FUNCTION_BLOCK FB_CamAxis
VAR
  _eCheck                       : E_CHECK_STATE;
  _nErrorId                     : UDINT; // datafield for Camming error

  _AxisSlave                    : REFERENCE TO AXIS_REF;
  _AxisMaster                   : REFERENCE TO AXIS_REF;

  _fbCamInV2                    : Tc2_MC2_Camming.MC_CamIn_V2;
  _fbScalingV2                  : Tc2_MC2_Camming.MC_CamScaling_V2;
  _fbCamInfoV2                  : Tc2_MC2_Camming.MC_CamInfo_V2;

  _fbReadMotionFunction         : Tc2_MC2_Camming.MC_ReadMotionFunction;
  _fbReadMotionFunctionPoint    : Tc2_MC2_Camming.MC_ReadMotionFunctionPoint;
  _fbReadMotionFunctionValues   : Tc2_MC2_Camming.MC_ReadMotionFunctionValues;

  _fbWriteMotionFunction        : Tc2_MC2_Camming.MC_WriteMotionFunction;
  _fbWriteMotionFunctionPoint   : Tc2_MC2_Camming.MC_WriteMotionFunctionPoint;


  _stCamInfoData                : Tc2_MC2_Camming.MC_CamInfoData;

END_VAR

METHOD CamInfo : E_PROGRESS
VAR_INPUT
  Execute           : BOOL;
  CamTableID        : Tc2_MC2_Camming.MC_CAM_ID;
  AtMasterPosition  : BOOL;
  MasterPosition    : LREAL;
END_VAR
VAR_INST
  _eState           : E_PROGRESS;
  _rValue           : LREAL;
  _udiErr           : UDINT;
  _stMsg            : ST_Message;
END_VAR
IF NOT Execute THEN _eState := E_PROGRESS.INIT; END_IF

CASE _eState
OF
  E_PROGRESS.INIT:
    IF Execute 
    THEN
      memset(ADR(_stMsg),0,SIZEOF(_stMsg));
      _udiErr                       := 0;
      _rValue                       := 0;
      _eState                       := E_PROGRESS.BUSY;

      _fbCamInfoV2(
              Slave                 := _AxisSlave, 
              Execute               := FALSE, 
              CamTableID            := CamTableID, 
              AtMasterPosition      := AtMasterPosition, 
              MasterPosition        := MasterPosition,
              CamInfo               => _stCamInfoData);
    END_IF
END_CASE
CASE _eState
OF
  E_PROGRESS.BUSY:
    _fbCamInfoV2(
              Slave                 := _AxisSlave, 
              Execute               := FALSE, 
              CamTableID            := CamTableID, 
              AtMasterPosition      := AtMasterPosition, 
              MasterPosition        := MasterPosition,
              CamInfo               => _stCamInfoData);

    IF (_fbCamInfoV2.Error)
    THEN
      _eState                       := E_PROGRESS.ERROR;
      _udiErr                       := _fbCamInfoV2.ErrorID;

      _stMsg.eType                  := E_MessageType.eMessageError;
      _stMsg.eDevice                := E_Device.Camming + TO_DINT(_AxisSlave.NcToPlc.AxisId);
      _stMsg.eSubdevice             := e_Subdevice.fbCamInfoV2;
      _stMsg.iErrorNumber           := _udiErr;
      f_MessageSet(_stMsg);

    ELSIF (_fbCamInfoV2.Done)
    THEN
      _eState                       := E_PROGRESS.READY;
    END_IF
END_CASE
CASE _eState
OF
  E_PROGRESS.STARTUP:
    _eState                         := E_PROGRESS.PREPARE;
END_CASE
CASE _eState
OF
  E_PROGRESS.PREPARE:
    _eState                         := E_PROGRESS.READY;
END_CASE
CASE _eState
OF
  E_PROGRESS.READY:
    _eState                         := E_PROGRESS.WAITING;
END_CASE
CASE _eState
OF
  E_PROGRESS.WAITING:
    _eState                         := E_PROGRESS.WORKING;
END_CASE
CASE _eState
OF
  E_PROGRESS.WORKING:
    _eState                         := E_PROGRESS.DONE;
END_CASE

CamInfo                             := _eState;
END_METHOD

METHOD PRIVATE CheckRef : BOOL
VAR_INPUT
END_VAR
IF NOT __ISVALIDREF(_AxisSlave)
THEN
  _eCheck                     := E_CHECK_STATE.CAM_SLAVE_AXIS_REF_INVALID;
  RETURN;
END_IF

IF NOT __ISVALIDREF(_AxisMaster)
THEN
  _eCheck                     := E_CHECK_STATE.CAM_MASTER_AXIS_REF_INVALID;
  RETURN;
END_IF

CheckRef                      := TRUE;
END_METHOD

METHOD Template : E_PROGRESS
VAR_INPUT
  Execute           : BOOL;
END_VAR
VAR_INST
  _eState           : E_PROGRESS;
  _rValue           : LREAL;
  _udiErr           : UDINT;
  _stMsg            : ST_Message;


END_VAR
IF NOT Check() THEN _eState := E_PROGRESS.ERROR; END_IF
IF NOT Execute THEN _eState := E_PROGRESS.INIT; END_IF

CASE _eState
OF
  E_PROGRESS.INIT:
    IF Execute 
    THEN
      memset(ADR(_stMsg),0,SIZEOF(_stMsg));
      _udiErr                       := 0;
      _rValue                       := 0;
      _eState                       := E_PROGRESS.BUSY;
    END_IF
END_CASE
CASE _eState
OF
  E_PROGRESS.BUSY:
    _eState                         := E_PROGRESS.STARTUP;
END_CASE
CASE _eState
OF
  E_PROGRESS.STARTUP:
    _eState                         := E_PROGRESS.PREPARE;
END_CASE
CASE _eState
OF
  E_PROGRESS.PREPARE:
    _eState                         := E_PROGRESS.READY;
END_CASE
CASE _eState
OF
  E_PROGRESS.READY:
    _eState                         := E_PROGRESS.WAITING;
END_CASE
CASE _eState
OF
  E_PROGRESS.WAITING:
    _eState                         := E_PROGRESS.WORKING;
END_CASE
CASE _eState
OF
  E_PROGRESS.WORKING:
    _eState                         := E_PROGRESS.DONE;
END_CASE

Template_1 := _eState;
END_METHOD

END_FUNCTION_BLOCK

(* stored: Version 1.1.0.1, ProductVersion 3.1.4024.12
   POU FB_CamAxis: Id {38a8250f-db6d-0d34-236a-d4cf6b05092d}, SpecialFunc None
   Folder methods: Id {1344f50f-5f72-04d5-3e8d-fe0c241daa85}
   Folder private: Id {40a64932-496b-0628-3ccd-b6d3e9fa789e}
   Method CamInfo: Id {144f8857-4ea4-0982-3c35-d07419e585c9}
   Method CheckRef: Id {3a0812aa-5da5-0fd3-0752-6798c438b735}
   Method Template: Id {daeae98d-95a2-0ae7-3740-aec6f888c178} *)
